{attribute 'qualified_only'}
{attribute 'strict'}
{attribute 'to_string'}
TYPE EnableState :
(
	Idle := 0,
    Reset_Movers := 10,
    Reset_Group := 20,
    Add_Mover := 30,
    Check_Add_Mover := 40,
    Enable_Movers := 50,
    Enable_Group := 60,
    Check_Standby := 70
);
END_TYPE

(* stored: Version 1.1.0.1
   DUT EnableState: Id {9e3b2163-4ed3-45c9-ada7-3fde7e08e450} *)
